FUNCTION sum : INT
VAR_INPUT
	num1 : INT;
	num2 : INT;
END_VAR
VAR
END_VAR

sum := num1 + num2;

END_FUNCTION

(* stored: Version 1.1.0.1, ProductVersion 3.1.4024.11
   POU sum: Id {e8fd35ca-d14c-4be9-8dc0-c7a15e5f49f2}, SpecialFunc None *)
